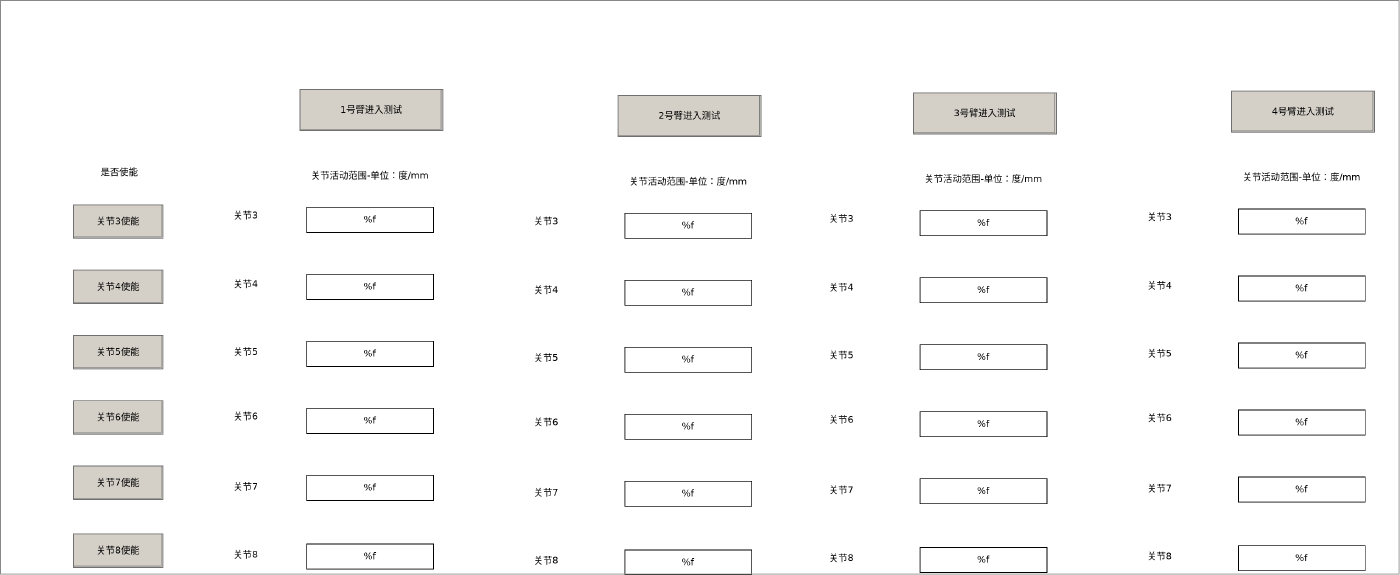
VISUALIZATION motRange_A1  // 1650x678
    Button (353,105 169x49), "1号臂进入测试", colour toggle: g_motionRangeTest.m_testMode[1]
        toggle g_motionRangeTest.m_testMode[1]
    Label (320,192 232x30), "关节活动范围-单位：度/mm"
    Label (217,240 145x28), "关节3"
    Label (217,321 145x28), "关节4"
    Label (217,401 145x28), "关节5"
    Label (217,477 145x28), "关节6"
    Label (217,560 145x28), "关节7"
    Label (217,640 145x28), "关节8"
    Rectangle (361,244 150x30), "%f", text variable: g_motionRangeTest.m_setupJntPosRange[1][3]
    Rectangle (361,323 150x30), "%f", text variable: g_motionRangeTest.m_setupJntPosRange[1][4]
    Rectangle (361,402 150x30), "%f", text variable: g_motionRangeTest.m_setupJntPosRange[1][5]
    Rectangle (361,481 150x30), "%f", text variable: g_motionRangeTest.m_slaveJntPosRange[1][1]
    Rectangle (361,560 150x30), "%f", text variable: g_motionRangeTest.m_slaveJntPosRange[1][2]
    Rectangle (361,641 150x30), "%f", text variable: g_motionRangeTest.m_slaveJntPosRange[1][3]
    Button (728,112 169x49), "2号臂进入测试", colour toggle: g_motionRangeTest.m_testMode[2]
        toggle g_motionRangeTest.m_testMode[2]
    Label (695,199 232x30), "关节活动范围-单位：度/mm"
    Label (571,247 145x28), "关节3"
    Label (571,328 145x28), "关节4"
    Label (571,408 145x28), "关节5"
    Label (571,484 145x28), "关节6"
    Label (571,567 145x28), "关节7"
    Label (571,647 145x28), "关节8"
    Rectangle (736,251 150x30), "%f", text variable: g_motionRangeTest.m_setupJntPosRange[2][3]
    Rectangle (736,330 150x30), "%f", text variable: g_motionRangeTest.m_setupJntPosRange[2][4]
    Rectangle (736,409 150x30), "%f", text variable: g_motionRangeTest.m_setupJntPosRange[2][5]
    Rectangle (736,488 150x30), "%f", text variable: g_motionRangeTest.m_slaveJntPosRange[2][1]
    Rectangle (736,567 150x30), "%f", text variable: g_motionRangeTest.m_slaveJntPosRange[2][2]
    Rectangle (736,648 150x30), "%f", text variable: g_motionRangeTest.m_slaveJntPosRange[2][3]
    Button (1076,109 169x49), "3号臂进入测试", colour toggle: g_motionRangeTest.m_testMode[3]
        toggle g_motionRangeTest.m_testMode[3]
    Label (1043,196 232x30), "关节活动范围-单位：度/mm"
    Label (919,244 145x28), "关节3"
    Label (919,325 145x28), "关节4"
    Label (919,405 145x28), "关节5"
    Label (919,481 145x28), "关节6"
    Label (919,564 145x28), "关节7"
    Label (919,644 145x28), "关节8"
    Rectangle (1084,248 150x30), "%f", text variable: g_motionRangeTest.m_setupJntPosRange[3][3]
    Rectangle (1084,327 150x30), "%f", text variable: g_motionRangeTest.m_setupJntPosRange[3][4]
    Rectangle (1084,406 150x30), "%f", text variable: g_motionRangeTest.m_setupJntPosRange[3][5]
    Rectangle (1084,485 150x30), "%f", text variable: g_motionRangeTest.m_slaveJntPosRange[3][1]
    Rectangle (1084,564 150x30), "%f", text variable: g_motionRangeTest.m_slaveJntPosRange[3][2]
    Rectangle (1084,645 150x30), "%f", text variable: g_motionRangeTest.m_slaveJntPosRange[3][3]
    Button (1451,107 169x49), "4号臂进入测试", colour toggle: g_motionRangeTest.m_testMode[4]
        toggle g_motionRangeTest.m_testMode[4]
    Label (1418,194 232x30), "关节活动范围-单位：度/mm"
    Label (1294,242 145x28), "关节3"
    Label (1294,323 145x28), "关节4"
    Label (1294,403 145x28), "关节5"
    Label (1294,479 145x28), "关节6"
    Label (1294,562 145x28), "关节7"
    Label (1294,642 145x28), "关节8"
    Rectangle (1459,246 150x30), "%f", text variable: g_motionRangeTest.m_setupJntPosRange[4][1]
    Rectangle (1459,325 150x30), "%f", text variable: g_motionRangeTest.m_setupJntPosRange[4][2]
    Rectangle (1459,404 150x30), "%f", text variable: g_motionRangeTest.m_setupJntPosRange[4][3]
    Rectangle (1459,483 150x30), "%f", text variable: g_motionRangeTest.m_slaveJntPosRange[4][1]
    Rectangle (1459,562 150x30), "%f", text variable: g_motionRangeTest.m_slaveJntPosRange[4][2]
    Rectangle (1459,643 150x30), "%f", text variable: g_motionRangeTest.m_slaveJntPosRange[4][3]
    Label (68,189 145x28), "是否使能"
    Button (86,241 106x40), "关节3使能", colour toggle: g_motionRangeTest.m_setupJntEnable[3]
        toggle g_motionRangeTest.m_setupJntEnable[3]
    Button (86,318 106x40), "关节4使能", colour toggle: g_motionRangeTest.m_setupJntEnable[4]
        toggle g_motionRangeTest.m_setupJntEnable[4]
    Button (86,395 106x40), "关节5使能", colour toggle: g_motionRangeTest.m_setupJntEnable[5]
        toggle g_motionRangeTest.m_setupJntEnable[5]
    Button (86,472 106x40), "关节6使能", colour toggle: g_motionRangeTest.m_slaveJntEnable[1]
        toggle g_motionRangeTest.m_slaveJntEnable[1]
    Button (86,549 106x40), "关节7使能", colour toggle: g_motionRangeTest.m_slaveJntEnable[2]
        toggle g_motionRangeTest.m_slaveJntEnable[2]
    Button (86,629 106x40), "关节8使能", colour toggle: g_motionRangeTest.m_slaveJntEnable[3]
        toggle g_motionRangeTest.m_slaveJntEnable[3]
END_VISUALIZATION

(* stored: Version 1.1.0.1, ProductVersion 3.1.4024.11
   Visu motRange_A1: Id {efca283f-21ae-4fe3-b194-d75e7dfc5bb7} *)
